FUNCTION_BLOCK TcoDataInspectorTests EXTENDS TcoInspectorTests
VAR
    _sut            : TcoInspectors.TcoDataInspector(THIS^, TcoCore.NO.Structure);
    _inspectedValue : STRING;
END_VAR

METHOD Inspect : TcoInspectors.IInspector
Inspect := _sut.Inspect(_inspectedValue);
END_METHOD

METHOD PROTECTED Main
SUPER^.Main();
END_METHOD

METHOD  WithCoordinator : REFERENCE TO TcoInspectorTests
VAR_INPUT
	inoCoordinator : TcoCore.ITcoCoordinator;
END_VAR
_sut.WithCoordinator(_coordinator);
WithCoordinator REF= THIS^;
END_METHOD

END_FUNCTION_BLOCK

(* stored: Version 1.1.0.1, ProductVersion 3.1.4024.9
   POU TcoDataInspectorTests: Id {7f0258dd-41d3-0c35-2a13-53089ff9ceff}, SpecialFunc None
   Method Inspect: Id {acc0c6bd-2e0e-0f04-3abe-e981b7b5da0f}
   Method Main: Id {98deef78-b00e-0980-0e31-8ab8d1c5e533}
   Method WithCoordinator: Id {5d47e5c3-93f1-0b7b-1be3-8f0136ba33a3} *)
